(* CODESYS project Eurowin_v_2_01_Final_PLC.project

Project tree, tasks and I/O mapping:
  Device : Owen SPK1xx, Owen, order no. 023, version 3.5.4.20
    application Application
      libraries: Standard, * (System); Util, * (System); VisuDialogs, * (System); ModulsOwenLib, 3.4.0.8 (Owen); CmpSysExec, 1.0.0.2 (Owen); SPK_Tools, 1.0.1 (Owen); Mx110Assistant, 3.5.4.0 (Owen)
      task MainTask (cyclic, interval t#20ms, priority 1) calls PLC_PRG
      task VISU_TASK (cyclic, interval 50 ms, priority 31) calls VisuElems.Visu_Prg
      program PLC_PRG [ST]: incrSpeed, decrSpeed, init, valveWork, lampsWork, getData, setData, modeCheck, pidReg, pidReg2, manualValveOff
      visualisation Main
      visualisation Alarm
      visualisation Parameters
      image pool ImagePool
      visualisation PidSettings
    Modbus_COM : Modbus COM, 3S - Smart Software Solutions GmbH, version 3.4.0.0
        settings: DataBits = 8; StopBits = 1; ComPort = 2
      Modbus_Master_COM_Port : Modbus Master, COM Port, 3S - Smart Software Solutions GmbH, version 3.5.5.0
          settings: Transmission = 'RTU'; ResponseTimeout = 300; TimeBetweenFrames = 10; Auto-restart communication = TRUE
        MU110_8I : MU110-8I, Owen, order no. 3.5.4.2, version 3.5.4.0
            settings: SlaveAddress = 1; ResponseTimeout = 300; UseExtendedFunctionCodes = TRUE
            unmapped channels: r.OE_1, in1, out1
        MV110_8A : MV110-8A, Owen, order no. 3.5.4.8, version 3.5.4.0
            settings: SlaveAddress = 17; ResponseTimeout = 300; UseExtendedFunctionCodes = TRUE
            unmapped channels: DP_1, in1, out1
        MU110_16R_K : MU110-16R_K, Owen, order no. 3.5.4.2, version 3.5.4.0
            settings: SlaveAddress = 33; ResponseTimeout = 300; UseExtendedFunctionCodes = TRUE
            unmapped channels: rMask, wMask, in1, out1
  text list GlobalTextList
  5ce3da45-db07-42e7-a21c-a00fff4ed8f6|D:\Pictures\ICONS\OnOff\off.png
  5ce3da45-db07-42e7-a21c-a00fff4ed8f6|D:\Pictures\ICONS\OnOff\on.png
*)

// Device/Application/PLC_PRG
PROGRAM PLC_PRG
VAR	
	blValve:BLINK;		
	
	iMaxSpeed:INT := 14;
	iMinSpeed:INT := 1;
	bInit:BOOL := TRUE;
	
	bKlapManOff1, bKlapManOff2, bKlapManOff3, bKlapManOff4 : BOOL;
	
	wsErrorMessage:WSTRING;
	iSpeed :INT;
	bRun, bRunAuto, bRunButton, bLamp1, bLamp2, bKlap1, bKlap2, bKlap3, bKlap4, bAlarmON, bAlarmOFF, bAlarmStarted, bAlrm1, bAlrm2, bAlrm3 :BOOL;
	rTemp1, rTemp2, rTemp3, rLampPwr1, rLampPwr2 : REAL;
END_VAR
VAR RETAIN
	rKoefON, rKoefOFF, rProfWidth :	REAL;	

	pid1:PID;
	rSET_POINT, rPidOut1, rKP, rTN, rTV, rY_MANUAL, rY_OFFSET, rY_MIN, rY_MAX : REAL;
	bMANUAL, bRESET, bLIMITS_ACTIVE, bOVERFLOW :BOOL;
	
	pid2:PID;
	rSET_POINT2, rPidOut2, rKP2, rTN2, rTV2, rY_MANUAL2, rY_OFFSET2, rY_MIN2, rY_MAX2 : REAL;
	bMANUAL2, bRESET2, bLIMITS_ACTIVE2, bOVERFLOW2 :BOOL;
	
	rTmpAlrm1, rTmpAlrm2, rTmpAlrm3, rTmpAlrmLow1, rTmpAlrmLow2, rTmpAlrmLow3: REAL;
END_VAR

init();
//
getData();
modeCheck();
valveWork();
lampsWork();

setData();

ACTION incrSpeed:
IF iSpeed < iMaxSpeed THEN
	iSpeed := iSpeed + 1;
END_IF
END_ACTION

ACTION decrSpeed:
IF iSpeed > iMinSpeed THEN
	iSpeed := iSpeed - 1;
END_IF
END_ACTION

ACTION init:
IF bInit THEN
	iSpeed := 1;
	rKoefOff:= 0.1;
	
	rY_MIN := 0;
	rY_MAX := 900;
	rSET_POINT := 50.0;
	rKP := 10.0;
	rTN := 5.0;
	rTV := 0.0;
	
	rY_MIN2 := 0;
	rY_MAX2 := 900;
	rSET_POINT2 := 50.0;
	rKP2 := 10.0;
	rTN2 := 5.0;
	rTV2 := 0.0;

	rTmpAlrm1 := 68;
	rTmpAlrm2 := 68;
	rTmpAlrm3 := 68;
	//
	bInit := FALSE;
END_IF
END_ACTION

ACTION valveWork:
IF bRun THEN
	IF rKoefOn <= 0 OR rKoefOff <= 0 THEN
		rKoefOn := 0.01;
		rKoefOff := 0.01;
	END_IF
	blValve(ENABLE := bRun, TIMEHIGH := REAL_TO_TIME(rProfWidth  * rKoefON), TIMELOW := REAL_TO_TIME((1000 * rKoefOFF)/ INT_TO_REAL(iSpeed)));
	bKlap1 := blValve.OUT AND blValve.ENABLE;
	bKlap2 := blValve.OUT AND blValve.ENABLE;
	bKlap3 := blValve.OUT AND blValve.ENABLE;
	bKlap4 := blValve.OUT AND blValve.ENABLE;
	manualValveOff();
	bRunAuto := TRUE;
END_IF
IF bRunAuto AND NOT bRun THEN
	bKlap1 := FALSE;
	bKlap2 := FALSE;
	bKlap3 := FALSE;
	bKlap4 := FALSE;
	bRunAuto := FALSE;
END_IF
END_ACTION

ACTION lampsWork:
IF bRun THEN
	pidReg();
	pidReg2();
	rLampPwr1 := pid1.Y / pid1.Y_MAX * 100;
	rLampPwr2 := pid2.Y / pid2.Y_MAX * 100;	
ELSE
	rPidOut1 := 0;
	rPidOut2 := 0;
	rLampPwr1 := 0;
	rLampPwr2 := 0;
END_IF
END_ACTION

ACTION getData:
rTemp1 := MV110_8A.rEAd_2;
rTemp2 := MV110_8A.rEAd_6;
rTemp3 := MV110_8A.rEAd_4;
END_ACTION

ACTION setData:
MU110_16R_K.wOut13 := bKlap1;
MU110_16R_K.wOut14 := bKlap2;
MU110_16R_K.wOut15 := bKlap3;
MU110_16R_K.wOut16 := bKlap4;

MU110_8I.rOE_1 := REAL_TO_WORD(rPidOut1);
MU110_8I.rOE_4 := REAL_TO_WORD(rPidOut2);
END_ACTION

ACTION modeCheck:
// Auto work off check
(*IF bRun AND NOT bRunButton THEN
	VisuElems.CURRENTVISU := 'Alarm';		
END_IF*)
IF bRunButton AND VisuElems.CURRENTVISU = 'Main' THEN
	bRun := TRUE;
END_IF
IF NOT bRunButton AND VisuElems.CURRENTVISU = 'Main' THEN
	bRun := FALSE;
END_IF

//Temp sensors check
IF MV110_8A.Stat_4 <> 0 THEN
		wsErrorMessage :=  "Нет связи с датчиком температуры входа профиля!";
END_IF
IF MV110_8A.Stat_6 <> 0 THEN
		wsErrorMessage :=  "Нет связи с датчиком температуры пленки!";
END_IF
IF MV110_8A.Stat_2 <> 0 THEN
		wsErrorMessage :=  "Нет связи с датчиком температуры выхода профиля!";
END_IF
IF MV110_8A.Stat_2 = 0 AND MV110_8A.Stat_4 = 0 AND MV110_8A.Stat_6 = 0 THEN
	wsErrorMessage := "";
END_IF
//Lamps condition indicator check
IF rLampPwr1 > 0 THEN
		bLamp1 := TRUE;
	ELSE
		bLamp1 := FALSE;
END_IF
IF rLampPwr2 > 0 THEN
		bLamp2 := TRUE;
	ELSE
		bLamp2 := FALSE;
END_IF

// Temp level check when running
IF rTemp1 > rTmpAlrm1 OR rTemp1 < rTmpAlrmLow1 THEN
	bAlrm1 := TRUE;
	ELSE
	bAlrm1 := FALSE;
END_IF
IF rTemp2 > rTmpAlrm2 OR rTemp2 < rTmpAlrmLow2 THEN
	bAlrm2 := TRUE;
	ELSE
	bAlrm2 := FALSE;
END_IF
IF rTemp3 > rTmpAlrm3 OR rTemp3 < rTmpAlrmLow3 THEN
	bAlrm3 := TRUE;
	ELSE
	bAlrm3 := FALSE;
END_IF

IF NOT bRun THEN
	bAlrm1 := FALSE;
	bAlrm2 := FALSE;
	bAlrm3 := FALSE;
END_IF

// Alarm sound initiation and termination
IF bAlrm1 OR bAlrm2 OR bAlrm3 THEN
	bAlarmON := TRUE;
	bAlarmStarted := TRUE;
END_IF
IF NOT bAlrm1 AND NOT bAlrm2 AND NOT bAlrm3 AND bAlarmStarted THEN
	bAlarmOFF := TRUE;
END_IF
IF bAlarmON THEN
	SysExecute('echo "1" > /sys/class/leds/pwm-beeper/brightness &');
	bAlarmON := FALSE;
END_IF
IF bAlarmOFF THEN
	SysExecute('echo "0" > /sys/class/leds/pwm-beeper/brightness &');
	bAlarmOFF := FALSE;
	bAlarmStarted := FALSE;
END_IF
END_ACTION

ACTION pidReg:
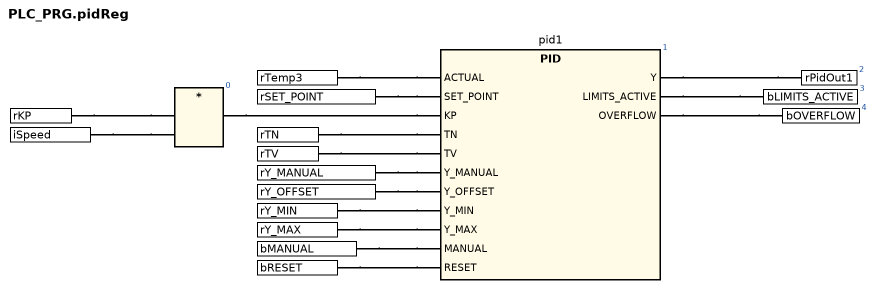
pid1(
    ACTUAL := rTemp3,
    SET_POINT := rSET_POINT,
    KP := rKP * iSpeed,
    TN := rTN,
    TV := rTV,
    Y_MANUAL := rY_MANUAL,
    Y_OFFSET := rY_OFFSET,
    Y_MIN := rY_MIN,
    Y_MAX := rY_MAX,
    MANUAL := bMANUAL,
    RESET := bRESET); // PID
rPidOut1 := pid1.Y;
bLIMITS_ACTIVE := pid1.LIMITS_ACTIVE;
bOVERFLOW := pid1.OVERFLOW;
END_ACTION

ACTION pidReg2:
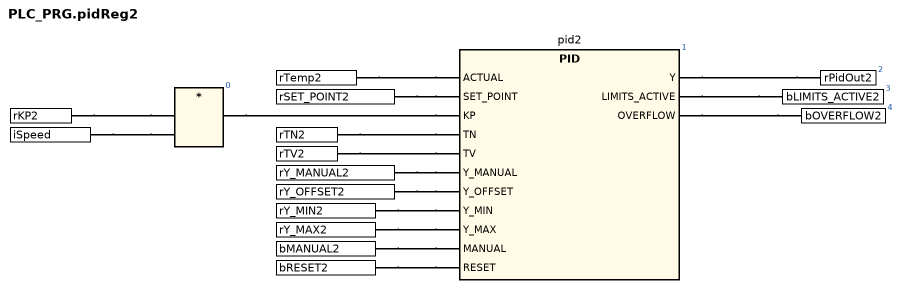
pid2(
    ACTUAL := rTemp2,
    SET_POINT := rSET_POINT2,
    KP := rKP2 * iSpeed,
    TN := rTN2,
    TV := rTV2,
    Y_MANUAL := rY_MANUAL2,
    Y_OFFSET := rY_OFFSET2,
    Y_MIN := rY_MIN2,
    Y_MAX := rY_MAX2,
    MANUAL := bMANUAL2,
    RESET := bRESET2); // PID
rPidOut2 := pid2.Y;
bLIMITS_ACTIVE2 := pid2.LIMITS_ACTIVE;
bOVERFLOW2 := pid2.OVERFLOW;
END_ACTION

ACTION manualValveOff:



IF bKlapManOff1 THEN
	bKlap1 := FALSE;
END_IF
IF bKlapManOff2 THEN
	bKlap2 := FALSE;
END_IF
IF bKlapManOff3 THEN
	bKlap3 := FALSE;
END_IF
IF bKlapManOff4 THEN
	bKlap4 := FALSE;
END_IF
END_ACTION

END_PROGRAM

// Device/Application/Main
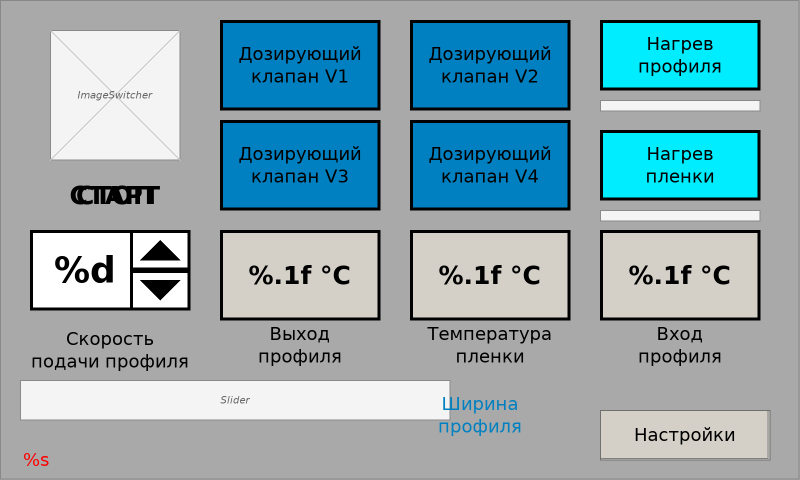
VISUALIZATION Main  // 800x480
    RoundedRectangle (600,20 160x70), "Нагрев профиля", colour toggle: PLC_PRG.bLamp1
        OnMouseClick:  ToggleVariable=PLC_PRG.bLamp1
    RoundedRectangle (600,130 160x70), "Нагрев пленки", colour toggle: PLC_PRG.bLamp2
        OnMouseClick:  ToggleVariable=PLC_PRG.bLamp2
    RoundedRectangle (30,230 110x80), "%d", text variable: PLC_PRG.iSpeed
    RoundedRectangle (220,20 160x90), "Дозирующий клапан V1", colour toggle: PLC_PRG.bKlap1
        OnMouseClick:  ToggleVariable=PLC_PRG.bKlap1
        OnMouseClick:  ToggleVariable=PLC_PRG.bKlapManOff1
    RoundedRectangle (220,230 160x90), "%.1f °C", text variable: PLC_PRG.rTemp1, colour toggle: PLC_PRG.bAlrm1
    RoundedRectangle (410,230 160x90), "%.1f °C", text variable: PLC_PRG.rTemp2, colour toggle: PLC_PRG.bAlrm2
    RoundedRectangle (600,230 160x90), "%.1f °C", text variable: PLC_PRG.rTemp3, colour toggle: PLC_PRG.bAlrm3
    RoundedRectangle (20,320 180x60), "Скорость подачи профиля"
    RoundedRectangle (220,320 160x50), "Выход профиля"
    RoundedRectangle (410,320 160x50), "Температура пленки"
    RoundedRectangle (600,320 160x50), "Вход профиля"
    RoundedRectangle (130,230 60x40)
        OnMouseClick: execute { PLC_PRG.incrSpeed(); }
    RoundedRectangle (130,270 60x40)
        OnMouseClick: execute { PLC_PRG.decrSpeed(); }
    Polygon (140,260) (160,240) (180,260)
        OnMouseClick: execute { PLC_PRG.incrSpeed(); }
    Polygon (140,280) (160,300) (180,280)
        OnMouseClick: execute { PLC_PRG.decrSpeed(); }
    RoundedRectangle (410,20 160x90), "Дозирующий клапан V2", colour toggle: PLC_PRG.bKlap2
        OnMouseClick:  ToggleVariable=PLC_PRG.bKlap2
        OnMouseClick:  ToggleVariable=PLC_PRG.bKlapManOff2
    RoundedRectangle (220,120 160x90), "Дозирующий клапан V3", colour toggle: PLC_PRG.bKlap3
        OnMouseClick:  ToggleVariable=PLC_PRG.bKlap3
        OnMouseClick:  ToggleVariable=PLC_PRG.bKlapManOff3
    RoundedRectangle (410,120 160x90), "Дозирующий клапан V4", colour toggle: PLC_PRG.bKlap4
        OnMouseClick:  ToggleVariable=PLC_PRG.bKlap4
        OnMouseClick:  ToggleVariable=PLC_PRG.bKlapManOff4
    RoundedRectangle (40,170 150x50), "СТАРТ", invisible if: PLC_PRG.bRun
    ImageSwitcher (50,30 130x130), variable: PLC_PRG.bRunButton, background image: ImagePool.off, image: ImagePool.on, behaviour: TOGGLE
    RoundedRectangle (40,170 150x50), "СТОП", invisible if: NOT PLC_PRG.bRun
    Button (600,410 170x50), "Настройки"
        OnMouseClick:  Assign=Parameters, Type=Assignment
    BarDisplayImage (600,100 160x11), value: PLC_PRG.rLampPwr1, style: BarDisplayImage-Green, scale format: %d, scale 0..100
    BarDisplayImage (600,210 160x11), value: PLC_PRG.rLampPwr2, style: BarDisplayImage-Green, scale format: %d, scale 0..100
    Rectangle (20,440 570x40), "%s", text variable: PLC_PRG.wsErrorMessage
    Slider (20,380 430x40), variable: PLC_PRG.rProfWidth, scale 0..100
    RoundedRectangle (220,20 160x90), colour toggle: PLC_PRG.bKlapManOff1
    RoundedRectangle (410,20 160x90), colour toggle: PLC_PRG.bKlapManOff2
    RoundedRectangle (220,120 160x90), colour toggle: PLC_PRG.bKlapManOff3
    RoundedRectangle (410,120 160x90), colour toggle: PLC_PRG.bKlapManOff4
    RoundedRectangle (420,390 120x50), "Ширина профиля"
END_VISUALIZATION

// Device/Application/Alarm
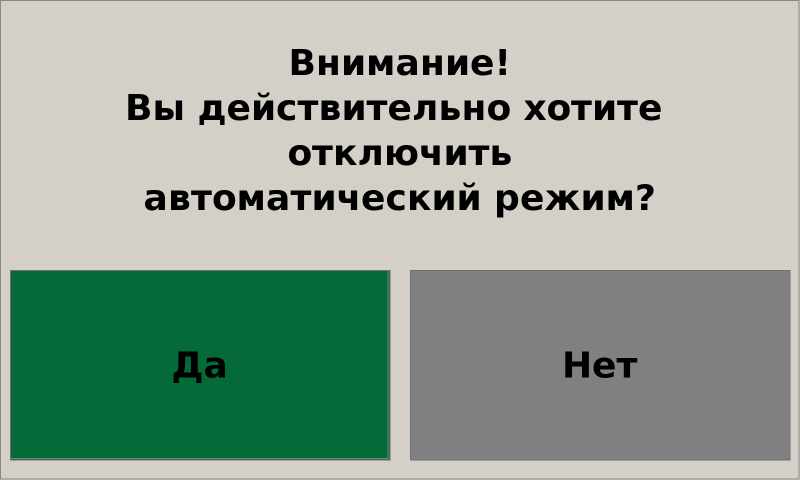
VISUALIZATION Alarm  // 800x480
    Rectangle (10,10 780x240), "Внимание! Вы действительно хотите отключить автоматический режим?"
    Button (10,270 380x190), "Да"
        OnMouseClick:  ToggleVariable=PLC_PRG.bRun
        OnMouseClick:  Assign=Main, Type=Assignment
    Button (410,270 380x190), "Нет"
        OnMouseClick:  Assign=Main, Type=Assignment
        OnMouseClick:  ToggleVariable=PLC_PRG.bRunButton
END_VISUALIZATION

// Device/Application/Parameters
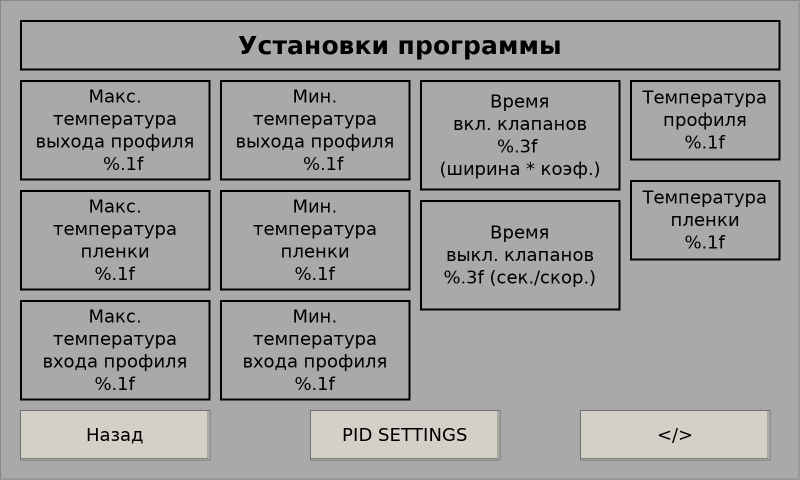
VISUALIZATION Parameters  // 800x480
    RoundedRectangle (20,80 190x100), "Макс. температура выхода профиля %.1f", text variable: PLC_PRG.rTmpAlrm1
        OnMouseClick: write the text variable via VisuDialogs.Numpad, min 0, max 100
    Button (20,410 190x50), "Назад"
        OnMouseClick:  Assign=Main, Type=Assignment
    RoundedRectangle (20,190 190x100), "Макс. температура пленки %.1f", text variable: PLC_PRG.rTmpAlrm2
        OnMouseClick: write the text variable via VisuDialogs.Numpad, min 0, max 100
    RoundedRectangle (20,300 190x100), "Макс. температура входа профиля %.1f", text variable: PLC_PRG.rTmpAlrm3
        OnMouseClick: write the text variable via VisuDialogs.Numpad, min 0, max 100
    RoundedRectangle (420,80 200x110), "Время вкл. клапанов %.3f (ширина * коэф.)", text variable: PLC_PRG.rKoefON
        OnMouseClick: write the text variable via VisuDialogs.Numpad, min 0, max 1000
    RoundedRectangle (420,200 200x110), "Время выкл. клапанов %.3f (сек./скор.)", text variable: PLC_PRG.rKoefOFF
        OnMouseClick: write the text variable via VisuDialogs.Numpad, min 0, max 100
    Button (580,410 190x50), "</>"
        OnMouseClick:  Type=Login
    RoundedRectangle (630,80 150x80), "Температура профиля %.1f", text variable: PLC_PRG.rSET_POINT
        OnMouseClick: write the text variable via VisuDialogs.Numpad, min 0, max 100
    RoundedRectangle (630,180 150x80), "Температура пленки %.1f", text variable: PLC_PRG.rSET_POINT2
        OnMouseClick: write the text variable via VisuDialogs.Numpad, min 0, max 100
    RoundedRectangle (20,20 760x50), "Установки программы"
    Button (310,410 190x50), "PID SETTINGS"
        OnMouseClick:  Assign=PidSettings, Type=Assignment
    RoundedRectangle (220,80 190x100), "Мин. температура выхода профиля %.1f", text variable: PLC_PRG.rTmpAlrmLow1
        OnMouseClick: write the text variable via VisuDialogs.Numpad, min 0, max 100
    RoundedRectangle (220,190 190x100), "Мин. температура пленки %.1f", text variable: PLC_PRG.rTmpAlrmLow2
        OnMouseClick: write the text variable via VisuDialogs.Numpad, min 0, max 100
    RoundedRectangle (220,300 190x100), "Мин. температура входа профиля %.1f", text variable: PLC_PRG.rTmpAlrmLow3
        OnMouseClick: write the text variable via VisuDialogs.Numpad, min 0, max 100
END_VISUALIZATION

// Device/Application/PidSettings
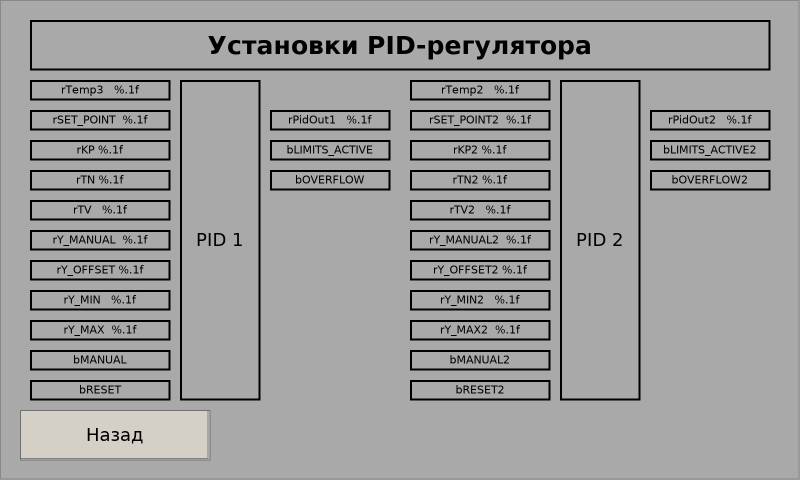
VISUALIZATION PidSettings  // 800x480
    RoundedRectangle (30,80 140x20), "rTemp3 %.1f", text variable: PLC_PRG.rTemp3
        OnMouseClick: write the text variable via VisuDialogs.Numpad, min 0, max 100
    Button (20,410 190x50), "Назад"
        OnMouseClick:  Assign=Main, Type=Previous
    RoundedRectangle (30,110 140x20), "rSET_POINT %.1f", text variable: PLC_PRG.rSET_POINT
        OnMouseClick: write the text variable via VisuDialogs.Numpad, min 0, max 100
    RoundedRectangle (30,170 140x20), "rTN %.1f", text variable: PLC_PRG.rTN
        OnMouseClick: write the text variable via VisuDialogs.Numpad
    RoundedRectangle (180,80 80x320), "PID 1"
    RoundedRectangle (30,20 740x50), "Установки PID-регулятора"
    RoundedRectangle (30,200 140x20), "rTV %.1f", text variable: PLC_PRG.rTV
        OnMouseClick: write the text variable via VisuDialogs.Numpad
    RoundedRectangle (30,230 140x20), "rY_MANUAL %.1f", text variable: PLC_PRG.rY_MANUAL
        OnMouseClick: write the text variable via VisuDialogs.Numpad
    RoundedRectangle (30,260 140x20), "rY_OFFSET %.1f", text variable: PLC_PRG.rY_OFFSET
        OnMouseClick: write the text variable via VisuDialogs.Numpad
    RoundedRectangle (30,290 140x20), "rY_MIN %.1f", text variable: PLC_PRG.rY_MIN
        OnMouseClick: write the text variable via VisuDialogs.Numpad
    RoundedRectangle (30,320 140x20), "rY_MAX %.1f", text variable: PLC_PRG.rY_MAX
        OnMouseClick: write the text variable via VisuDialogs.Numpad
    RoundedRectangle (30,350 140x20), "bMANUAL", colour toggle: PLC_PRG.bMANUAL
        OnMouseClick:  ToggleVariable=PLC_PRG.bMANUAL
    RoundedRectangle (30,380 140x20), "bRESET", colour toggle: PLC_PRG.bRESET
        OnMouseClick:  ToggleVariable=PLC_PRG.bRESET
    RoundedRectangle (270,110 120x20), "rPidOut1 %.1f", text variable: PLC_PRG.rPidOut1
    RoundedRectangle (270,140 120x20), "bLIMITS_ACTIVE", colour toggle: PLC_PRG.bLIMITS_ACTIVE
    RoundedRectangle (270,170 120x20), "bOVERFLOW", colour toggle: PLC_PRG.bOVERFLOW
    RoundedRectangle (30,140 140x20), "rKP %.1f", text variable: PLC_PRG.rKP
        OnMouseClick: write the text variable via VisuDialogs.Numpad
    RoundedRectangle (410,80 140x20), "rTemp2 %.1f", text variable: PLC_PRG.rTemp2
        OnMouseClick: write the text variable via VisuDialogs.Numpad, min 0, max 100
    RoundedRectangle (410,110 140x20), "rSET_POINT2 %.1f", text variable: PLC_PRG.rSET_POINT2
        OnMouseClick: write the text variable via VisuDialogs.Numpad, min 0, max 100
    RoundedRectangle (410,170 140x20), "rTN2 %.1f", text variable: PLC_PRG.rTN2
        OnMouseClick: write the text variable via VisuDialogs.Numpad
    RoundedRectangle (560,80 80x320), "PID 2"
    RoundedRectangle (410,200 140x20), "rTV2 %.1f", text variable: PLC_PRG.rTV2
        OnMouseClick: write the text variable via VisuDialogs.Numpad
    RoundedRectangle (410,230 140x20), "rY_MANUAL2 %.1f", text variable: PLC_PRG.rY_MANUAL2
        OnMouseClick: write the text variable via VisuDialogs.Numpad
    RoundedRectangle (410,260 140x20), "rY_OFFSET2 %.1f", text variable: PLC_PRG.rY_OFFSET2
        OnMouseClick: write the text variable via VisuDialogs.Numpad
    RoundedRectangle (410,290 140x20), "rY_MIN2 %.1f", text variable: PLC_PRG.rY_MIN2
        OnMouseClick: write the text variable via VisuDialogs.Numpad
    RoundedRectangle (410,320 140x20), "rY_MAX2 %.1f", text variable: PLC_PRG.rY_MAX2
        OnMouseClick: write the text variable via VisuDialogs.Numpad
    RoundedRectangle (410,350 140x20), "bMANUAL2", colour toggle: PLC_PRG.bMANUAL2
        OnMouseClick:  ToggleVariable=PLC_PRG.bMANUAL
    RoundedRectangle (410,380 140x20), "bRESET2", colour toggle: PLC_PRG.bRESET2
        OnMouseClick:  ToggleVariable=PLC_PRG.bRESET
    RoundedRectangle (650,110 120x20), "rPidOut2 %.1f", text variable: PLC_PRG.rPidOut2
    RoundedRectangle (650,140 120x20), "bLIMITS_ACTIVE2", colour toggle: PLC_PRG.bLIMITS_ACTIVE2
    RoundedRectangle (650,170 120x20), "bOVERFLOW2", colour toggle: PLC_PRG.bOVERFLOW2
    RoundedRectangle (410,140 140x20), "rKP2 %.1f", text variable: PLC_PRG.rKP2
        OnMouseClick: write the text variable via VisuDialogs.Numpad
END_VISUALIZATION
